Staubli VAL3: OnEvent1.pgx

program OnEvent1()
  local bool l_bRes
begin
  //-----------------------------------------------------------------------
  //Header begin
  //LasMAN3.7
  //Description of program
  //
  //Input parameters
  //
  //Output paramaters
  //Example
  //  call OnEvent1()
  //History
  //  Creation : 2013-06-23  y.ye@staubli.com
  //Header end
  //-----------------------------------------------------------------------

  DataBase:bStopPoll=true
  call TxtFile:ReadCfg(l_bRes)
  IO:bWeldEnable=TxtFile:bWeldEnable
  IO:bWeldEnable=TxtFile:bWeldEnable
  IO:bExt7AxisEnable=TxtFile:b7Axis
  IO:bExt8AxisEnable=TxtFile:b8Axis
  DataBase:bStopPoll=false

  if l_bRes

    call Kit:GoHome()
  else
    popUpMsg("读取配置文件出错")
  endIf
  DataBase:nInterfaceType=9
end
